(* PLC project Generated.project, CODESYS CODESYS V3.5 SP19 Patch 1 *)
(* stored: creationDateTime 2026-11-18T10:48:20.644928, modificationDateTime 2026-11-18T10:48:20.644928 *)

(* ═══════════════════════════════════════════════════════════════ 🚦 ST_WinchState — États, mesures et diagnostics HMI pour un Treuil M1/M2 ─────────────────────────────────────────────────────────────── 🎨 Destiné aux retours d'informations et bargraphes HMI. ═══════════════════════════════════════════════════════════════ *)
TYPE ST_WinchState : STRUCT
  Position_M : REAL;  (* 🚦 États & Mesures (Lecture seule) 📊 Position actuelle du câble (mètres) *)
  MeasuredSpeed_Mps : REAL;  (* 📏 Vitesse linéaire mesurée du câble (m/s), valeur absolue *)
  SpeedDelta_Mps : REAL;  (* 🔍 Variation de vitesse entre deux scans (m/s) *)
  SpeedVariationDetected : BOOL;  (* 🔍 Seuil de variation dépassé sur le scan courant *)
  SpeedVariationConfirmed : BOOL;  (* 🛡️ Variation confirmée pendant la durée paramétrée *)
  SpeedStable : BOOL;  (* 🟢 Vitesse stable pendant la durée paramétrée *)
  SpeedMonitorError : BOOL;  (* Défaut mémorisé du moniteur vitesse *)
  SpeedMonitorErrorId : WORD;  (* ❌ Bitfield du moniteur vitesse *)
  EstimatedLoadPct : REAL;  (* 📊 Estimation empirique, non certifiée *)
  LoadEstimateConfigured : BOOL;  (* 🟢 Table charge validée pour lecture *)
  SpeedGuardLimited : BOOL;  (* 🛡️ Palier limité par vitesse réelle *)
  SpeedCmd_Pct : REAL;  (* 📈 Commande de vitesse finale après rampe (%) *)
  StepNumber : INT;  (* 🔢 Palier de vitesse actif (0..5) *)
  FBState : E_State;  (* 🤖 État de l'automate interne (FB_Winch) *)
  AxisBlockReason : E_WinchTraceBlockReason;  (* 🧩 Cause prioritaire de blocage (miroir de TraceMx.BlockReason) *)
  Ready : BOOL;  (* 🟢 Treuil prêt à fonctionner *)
  Busy : BOOL;  (* ⚙️ Mouvement en cours *)
  Done : BOOL;  (* ✅ Action terminée *)
  Error : BOOL;  (* Treuil en défaut *)
  ErrorId : WORD;  (* ❌ Code bitfield du défaut treuil *)
  FaultLatched : BOOL;  (* 🔒 Défaut treuil latché (acquittable Reset) *)
  RelayFwd : BOOL;  (* 🔌 Sorties Physiques / Indicateurs LEDs 🛗 Relais Ascending activé *)
  RelayRev : BOOL;  (* 🛗 Relais Descending activé *)
  Contactor1 : BOOL;  (* 🔌 Contacteur vitesse palier 1 *)
  Contactor2 : BOOL;  (* 🔌 Contacteur vitesse palier 2 *)
  Contactor3 : BOOL;  (* 🔌 Contacteur vitesse palier 3 *)
  Contactor4 : BOOL;  (* 🔌 Contacteur vitesse palier 4 *)
  BrakeCmd : BOOL;  (* 🔓 Commande frein (TRUE = desserré / libre) *)
  FinalInterlockState : E_WinchFinalInterlockState;  (* 🛡️ État final lecture seule *)
  FinalInterlockReason : E_WinchFinalInterlockReason;  (* 🛡️ Cause finale mémorisée *)
  FinalInterlockError : BOOL;  (* 🛡️ Défaut final mémorisé *)
  FinalInterlockErrorId : WORD;  (* 🛡️ Bitfield final *)
  FinalRestartInhibit : BOOL;  (* 🔒 Reset + neutre + nouvelle demande obligatoires *)
  FinalRestartRequired : BOOL;  (* 🔒 Purge anti-redemarrage armee : AuthorizedStep force a 0 tant que non purgee (distinct de RestartInhibit) *)
  FinalMotorRequest : BOOL;  (* 🔒 Demande moteur vue par la barriere finale (palier>0 ET un seul sens) *)
  FinalNeutralRequestSeen : BOOL;  (* 🔒 Passage au neutre observe pendant un RestartInhibit *)
  BrakeCommandOpenConfirmed : BOOL;  (* 🔌 Contacteur/bobine desserrage confirmé, pas frein mécanique *)
  FinalAuthorizedStep : INT;  (* 🪜 Palier réellement autorisé *)
  FinalBrakeTimeoutElapsed : TIME;  (* ⏱️ Écoulé watchdog 500ms *)
  FinalRestartDelayElapsed : TIME;  (* ⏱️ Écoulé verrou redémarrage 900ms *)
  FinalStepDelayElapsed : TIME;  (* ⏱️ Écoulé entre paliers 1s250 *)
  Encoder : ST_EncoderHMI;  (* 🛡️ Sécurités & Diagnostics 🧲 Données d'échange et diagnostic du codeur — porte aussi les 9 champs Homing* (voir ST_EncoderHMI) *)
  ContactorsCheck : ST_ContactorCheck;  (* 🔍 Diagnostics de cohérence contacteurs réutilisés 🔌 Coherence contacteurs sens+vitesse *)
  BrakeContactorCheck : ST_ContactorCheck;  (* 🔌 Coherence retour frein *)
  InhibitActive : BOOL;  (* miroir lecture seule — inhibition arbitrée *)
  BottomLimitActiveM : REAL;  (* 🐢 : ralentissement sur bordure — diagnostic zone/limite active 📏 Limite basse active (m) — câble physique OU légale, la plus restrictive *)
  InTopSlowdownZone : BOOL;  (* 🐢 Palier plafonné à 1 : approche limite haute *)
  InBottomSlowdownZone : BOOL;  (* 🐢 Palier plafonné à 1 : approche limite basse (câble ou légale) *)
  CommandedAscent : BOOL;  (* 🩺 Diagnostic délai ressenti à la remontée 🩺 Sens interne mémorisé FB_Winch : montée *)
  CommandedDescend : BOOL;  (* 🩺 Sens interne mémorisé FB_Winch : descente *)
  DirectionChangeDelayElapsed : TIME;  (* 🩺 Écoulé de l'interlock changement/reprise de sens *)
  DirectionChangePending : BOOL;  (* 🩺 TRUE tant que CommandedDirection n'a pas rejoint Direction *)
END_STRUCT;
END_TYPE

(* values of E_State: DISABLED: Enable faux, neutralisé; INIT: Démarrage / vérifs; READY: Prêt, attend ordre; BUSY: Action en cours; DONE: Action terminée; STOPPING: Décél rampe avant arrêt (StartStop=FALSE ou SafeStop=TRUE); ERROR: Défaut actif non acquitté (FB en erreur — HMI non aveugle) *)

{attribute 'qualified_only'}
{attribute 'strict'}
TYPE E_State : (DISABLED := 0, INIT := 1, READY := 2, BUSY := 3, DONE := 4, STOPPING := 5, ERROR := 6);
END_TYPE

(* values of E_WinchFinalInterlockReason: NONE: Aucun blocage actif; BRAKE_COMMAND_NOT_CONFIRMED: Absence confirmation ouverture frein > 500ms; RESTART_INHIBITED: Inhibition redemarrage actif; SENSE_DROP_TIMEOUT: T_max §3bis depasse sans confirmation retombee (AC7) *)

{attribute 'qualified_only'}
{attribute 'strict'}
TYPE E_WinchFinalInterlockReason : (NONE := 0, BRAKE_COMMAND_NOT_CONFIRMED := 1, RESTART_INHIBITED := 2, SENSE_DROP_TIMEOUT := 3);
END_TYPE

(* values of E_WinchFinalInterlockState: DISABLED: Desactive / Hors service; READY: Pret / Etat nominal; WAIT_BRAKE_COMMAND_CONFIRMATION: Attente confirmation feedback frein; WAIT_STEP_DELAY: Temporisation changement de palier; WAIT_RESTART_DELAY: Temporisation anti-court-cycle redemarrage; FAULT: Etat de defaut; WAIT_SENSE_DROP_CONFIRM: Maintien §3bis du contacteur de sens (AC6/AC7) *)

{attribute 'qualified_only'}
{attribute 'strict'}
TYPE E_WinchFinalInterlockState : (DISABLED := 0, READY := 1, WAIT_BRAKE_COMMAND_CONFIRMATION := 2, WAIT_STEP_DELAY := 3, WAIT_RESTART_DELAY := 4, FAULT := 5, WAIT_SENSE_DROP_CONFIRM := 6);
END_TYPE

(* values of E_WinchTraceBlockReason: NONE: Aucun blocage - au moins un sens effectivement permis; POWER_CUTOFF: Coupure puissance amont (instSafetyWinch.PowerCutOff) - priorite max; AXIS_DISABLED: Axe neutralise (Mode=DISABLE ou InhibitMx -> Enable FALSE); SAFESTOP: SafeStop effectif (rampe rapide demandee); SAFETY_FAULT: Defaut safety latched (FB_Safety_Winch.Fault.Error); SAFETY_PERMIT_MISSING: Aucun sens ne delivre de permit safety (limite / mou de cable / homing); PROCESS_PERMIT_MISSING: Permit process absent (benne / fond Kobold / limite legale / extraction); COUPLING_BLOCKED: Couplage synchro anti-telescopage (l'autre axe bloque); WINCH_FAULT: Defaut treuil latched (FB_Winch.Fault.Error); FINAL_INTERLOCK_BLOCKED: Barriere finale en defaut (frein / redemarrage) *)

{attribute 'qualified_only'}
{attribute 'strict'}
TYPE E_WinchTraceBlockReason : (NONE := 0, POWER_CUTOFF := 1, AXIS_DISABLED := 2, SAFESTOP := 3, SAFETY_FAULT := 4, SAFETY_PERMIT_MISSING := 5, PROCESS_PERMIT_MISSING := 6, COUPLING_BLOCKED := 7, WINCH_FAULT := 8, FINAL_INTERLOCK_BLOCKED := 9);
END_TYPE

(* ======================================================================= 🔌 ST_ContactorCheck — Double vérification commande/retour contacteur ─────────────────────────────────────────────────────────────── 🎯 Rôle : Structure de diagnostic pour vérification commande vs retour 📊 Diagnostic : Détection des défauts contacteur (StuckClosed / StuckOpen) 📄 Doc métier : DOC/AF/AF_Partie-03_Contrats_Composants_v2.3.md §2 ======================================================================= *)
TYPE ST_ContactorCheck : STRUCT
  Command : BOOL;  (* Ordre envoyé au contacteur (TRUE = fermé/actif) *)
  Feedback : BOOL;  (* Retour d'état câblé (TRUE = effectivement fermé) *)
  StuckClosed : BOOL;  (* Diag : commande OFF mais retour ON depuis trop longtemps → PowerCutOff *)
  StuckOpen : BOOL;  (* Diag : commande ON mais retour OFF depuis trop longtemps *)
END_STRUCT;
END_TYPE

(* ═══════════════════════════════════════════════════════════════ 🧲 ST_EncoderHMI — Données d'échange IHM pour les codeurs absolus ─────────────────────────────────────────────────────────────── 🎨 Destiné à l'affichage des informations et diagnostics des codeurs. ═══════════════════════════════════════════════════════════════ *)
TYPE ST_EncoderHMI : STRUCT
  RawPos : UDINT;  (* 📊 Position brute lue sur le bus *)
  Alarms : UINT;  (* ⚠️ Code d'alarme brut du codeur *)
  Warnings : UINT;  (* 🟧 Code d'avertissement brut du codeur *)
  SlaveOperational : BOOL;  (* 📡 Esclave EtherCAT opérationnel *)
  PresetTriggerCmd : WORD;  (* 🎯 Commande de preset active *)
  PresetValueOut : UDINT;  (* 📐 Valeur de preset envoyée au codeur *)
  Error : BOOL;  (* Codeur en défaut (liaison EtherCAT ou preset) *)
  ErrorId : WORD;  (* ❌ Code défaut codeur *)
  Homed : BOOL;  (* 🎯 Homing — prise d'origine / référencement 🎯 Prise d'origine (Homing) validée *)
  HomingBusy : BOOL;  (* ⏳ Référencement en cours *)
  HomingDone : BOOL;  (* ✅ Pulse de référencement réussi *)
  HomingError : BOOL;  (* Défaut de référencement *)
  HomingErrorId : WORD;  (* ❌ Bitfield défaut homing *)
  HomingState : E_State;  (* 🤖 État FB_Encoder_Homing *)
  HomingStateAtError : E_State;  (* 🧭 État lors du défaut *)
  HomingSuspect : BOOL;  (* ⚠️ Référence à confirmer *)
  HomingRefRaw : UDINT;  (* 📐 Référence brute appliquée *)
END_STRUCT;
END_TYPE
